TYPE ST_ChamberAlarm :
STRUCT
	dtTime:STRING(255);
	sAlarmText:STRING(255);
	
	
END_STRUCT
END_TYPE

(* stored: Version 1.1.0.1, ProductVersion 3.1.4022.16
   DUT ST_ChamberAlarm: Id {21d86930-5b9c-4a7d-821f-00af54f2eaad} *)
